//-----------------------------------------------------------------------------------------
//
//                  				ST_Tool_Corrector_M
//
//								Structure correcteur M outil 			
//-----------------------------------------------------------------------------------------
//
//Auteur: G.GOETZ (inspired by S.FLEURY)
//Création: 20.01.2026
//Dernière modification : 20.01.2026 (G.GOETZ)
//       			
//-----------------------------------------------------------------------------------------
//
//     							Liste des modifications  	
//
// 20.01.2026 (G.GOETZ) -> Création		
//-----------------------------------------------------------------------------------------

TYPE ST_Tool_Corrector_M :
STRUCT
	
	(** SETUP DINT **)
		Longueur : DINT ;
		UsureLongueur : DINT ;
		Rayon : DINT ;
		UsureRayon : DINT ;
		PositionW : DINT ;
		
END_STRUCT
END_TYPE

(* stored: Version 1.1.0.1, ProductVersion 3.1.4026.17
   DUT ST_Tool_Corrector_M: Id {dfff8b5c-f022-4e38-9e01-4f8fc8f264a1} *)
